// TwinCAT 3 PLC project PLCStudent
// ProgramVersion: 3.1.4026.13
// libraries:
//   Tc2_Standard, * (Beckhoff Automation GmbH)
//   Tc2_System, * (Beckhoff Automation GmbH)
//   Tc3_Module, * (Beckhoff Automation GmbH)
// project tree:
//   / PlcTask.TcTTO (not stored)
//   POUs/ MAIN.TcPOU, Control_FBD.TcPOU
// (motion and I/O tree: see PLC project plcsim)
// real-time tasks:
//   TASK PlcTask: cycle T#80ms, priority 1, ADS port 350
//   TASK PlcTask1: cycle T#10ms, priority 20, ADS port 351
// variable links:
//   PLCSim/PLCSim Instance <-> PLCStudent/PLCStudent Instance
//     PlcTask Inputs/GVL.ixBack <-> PlcTask Outputs/Control_FBD.qxBack
//     PlcTask Inputs/GVL.ixDispBit1 <-> PlcTask Outputs/Control_FBD.qxDispBit1
//     PlcTask Inputs/GVL.ixDispBit2 <-> PlcTask Outputs/Control_FBD.qxDispBit2
//     PlcTask Inputs/GVL.ixDrain <-> PlcTask Outputs/Control_FBD.qxDrain
//     PlcTask Inputs/GVL.ixFill <-> PlcTask Outputs/Control_FBD.qxFill
//     PlcTask Inputs/GVL.ixForw <-> PlcTask Outputs/Control_FBD.qxForw
//     PlcTask Inputs/GVL.ixHeat <-> PlcTask Outputs/Control_FBD.qxHeat
//     PlcTask Inputs/GVL.ixSpin <-> PlcTask Outputs/Control_FBD.qxSpin
//     PlcTask Outputs/GVL.qxLevel1 <-> PlcTask Inputs/Control_FBD.ixLevel1
//     PlcTask Outputs/GVL.qxLevel2 <-> PlcTask Inputs/Control_FBD.ixLevel2
//     PlcTask Outputs/GVL.qxLevel3 <-> PlcTask Inputs/Control_FBD.ixLevel3
//     PlcTask Outputs/GVL.qxNotEmpty <-> PlcTask Inputs/Control_FBD.ixNotEmpty
//     PlcTask Outputs/GVL.qxPulse <-> PlcTask Inputs/Control_FBD.ixPulse
//     PlcTask Outputs/GVL.qxSetLevel <-> PlcTask Inputs/Control_FBD.ixSetLevel
//     PlcTask Outputs/GVL.qxStart <-> PlcTask Inputs/Control_FBD.ixStart
//     PlcTask Outputs/GVL.qxTempOk <-> PlcTask Inputs/Control_FBD.ixTempOk

// ---- POUs/MAIN.TcPOU
PROGRAM MAIN
VAR
END_VAR

Control_FBD();

END_PROGRAM

// ---- POUs/Control_FBD.TcPOU
PROGRAM Control_FBD
VAR
	
	ixPulse			AT %I*:	BOOL; 		(* PULS button *)
	ixStart			AT %I*:	BOOL; 		(* START switch *)
	ixSetLevel		AT %I*:	BOOL; 		(* NIVÅ switch *)
	ixLevel3		AT %I*:	BOOL; 		(* Sensor for level 3 *)
	ixLevel2		AT %I*:	BOOL; 		(* Sensor for level 2 *)
	ixLevel1		AT %I*:	BOOL; 		(* Sensor for level 1 *)
	ixNotEmpty		AT %I*:	BOOL; 		(* Sensor for not empty *)
	ixTempOk		AT %I*:	BOOL; 		(* Temp sensor *)

	qxForw			AT %Q*:	BOOL; 		(* Washer cylinder forward *)
	qxBack			AT %Q*:	BOOL; 		(* Washer cylinder back *)
	qxSpin			AT %Q*:	BOOL; 		(* Hi-spin/Centrifuge need qxForw or qxBack*)
	qxFill			AT %Q*:	BOOL; 		(* Fill water *)
	qxDrain			AT %Q*:	BOOL; 		(* Drain water *)
	qxHeat			AT %Q*:	BOOL; 		(* Heat water *)
	qxDispBit1		AT %Q*:	BOOL; 		(* Display bit 1 *)
	qxDispBit2		AT %Q*:	BOOL; 		(* Display bit 2 *)
	// local variables
	mxFill: BOOL;
	tpForw: TP; //Timer Pulse Forward
	mxForw: BOOL;
	Steps: INT;
	tpBack: TP; // Timer Pulse backward
	mxBack: BOOL;
	tpDry: TP;
	mxDry: BOOL;
	TP_Forw: BOOL;
	mxDrain: BOOL;
	TP_Back: BOOL;
	mxSpin: BOOL;
END_VAR

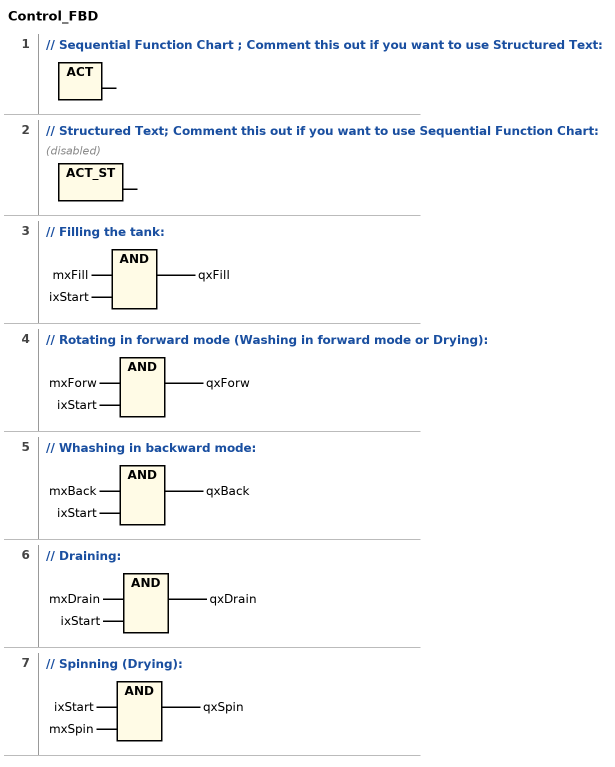
// NETWORK 1
// label: // Sequential Function Chart ; Comment this out if you want to use Structured Text
ACT();

// NETWORK 2 (disabled)
// label: // Structured Text; Comment this out if you want to use Sequential Function Chart
// ACT_ST();

// NETWORK 3
// label: // Filling the tank
qxFill := mxFill AND ixStart;

// NETWORK 4
// label: // Rotating in forward mode (Washing in forward mode or Drying)
qxForw := mxForw AND ixStart;

// NETWORK 5
// label: // Whashing in backward mode
qxBack := mxBack AND ixStart;

// NETWORK 6
// label: // Draining
qxDrain := mxDrain AND ixStart;

// NETWORK 7
// label: // Spinning (Drying)
qxSpin := ixStart AND mxSpin;

ACTION ACT:
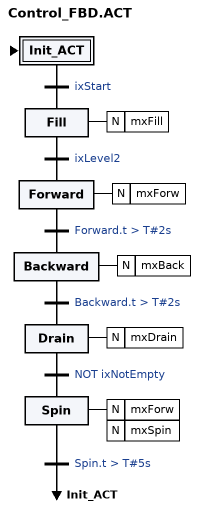
INITIAL_STEP Init_ACT:
END_STEP
TRANSITION FROM Init_ACT TO Fill
    := ixStart;
END_TRANSITION
STEP Fill:
    mxFill(N);
END_STEP
TRANSITION FROM Fill TO Forward
    := ixLevel2;
END_TRANSITION
STEP Forward:
    mxForw(N);
END_STEP
TRANSITION FROM Forward TO Backward
    := Forward.t > T#2s;
END_TRANSITION
STEP Backward:
    mxBack(N);
END_STEP
TRANSITION FROM Backward TO Drain
    := Backward.t > T#2s;
END_TRANSITION
STEP Drain:
    mxDrain(N);
END_STEP
TRANSITION FROM Drain TO Spin
    := NOT ixNotEmpty;
END_TRANSITION
STEP Spin:
    mxForw(N);
    mxSpin(N);
END_STEP
TRANSITION FROM Spin TO Init_ACT
    := Spin.t > T#5s;
END_TRANSITION
END_ACTION

ACTION ACT_ST:
CASE Steps OF
	0:	// Fill the tank if the machine is in start mode and empty
		IF ixStart THEN
			IF ixLevel2 = FALSE THEN
				mxFill := TRUE;
			ELSE
				mxFill := FALSE;
				Steps := 1;
			END_IF
		END_IF
	1:  (*
			Wash in forward mode for two seconds if
				1. The machine is in start mode
				2. The tank is filled up to level 2
		*)
		tpForw(IN := TRUE, PT:= T#2S);
		TP_Forw := tpForw.Q;
		IF TP_forw THEN
			mxForw := TRUE;
		ELSE
			mxForw := FALSE;
			tpForw(IN := FALSE);
			Steps := 2;
		END_IF
		
	2:  (*
			Wash for another two seconds in backward mode if
				1. The machine is in start mode
				2. The tank is filled up to level 2
				3. Washing has already been done in froward mode for two seconds
		*)
		tpBack(IN := TRUE, PT:= T#2S);
		TP_Back := tpBack.Q;
		IF TP_Back THEN
			mxBack := TRUE;
		ELSE
			mxBack := FALSE;
			tpBack(IN := FALSE);
			Steps := 3;
		END_IF

	3:  (*
			Drain the tank if
				1. The machine is in start mode
				2. The tank is not empty
				3. Washing has already been done.
		*)
	    IF ixNotEmpty THEN
			mxDrain := TRUE;
		ELSE
			mxDrain := FALSE;
			Steps := 4;
		END_IF
	
	4:  (*
			Drying: Spin the container in forward mode
				1. The machine is in start mode
				2. The tank is empty
				3. Washing and Draining have already been done.
		*)
		tpDry(IN := TRUE, PT:= T#5S);
		mxDry := tpDry.Q;
		IF mxDry THEN
			mxForw := TRUE;
			mxSpin := TRUE;
		ELSE
			mxForw := FALSE;
			mxSpin := FALSE;
			tpDry(IN := FALSE);
			Steps := 0;
		END_IF
		
END_CASE
END_ACTION

END_PROGRAM
